KUKA KRL program: PrintBool.src

&ACCESS RVO
&PARAM EDITMASK = *
DEF PrintBool(name[]:in, value:in )
decl bool value
decl char name[]
decl KrlMsg_T msg
decl KrlMsgPar_T par[3]
decl KrlMsgOpt_T opt
decl int handle

msg = {modul[] "print", Nr 1, msg_txt[] "<bool> %1 = %2"}
par[1] = {par_type #value, par_txt[] " "}
par[1].par_txt[] = name[]
if value==true then
 par[2] = {par_type #value, par_txt[] "true"}
else
 par[2] = {par_type #value, par_txt[] "false"}
endif
opt = {vl_stop true, clear_p_reset true, clear_p_SAW false, log_to_DB false}
handle = Set_KrlMsg (#notify, msg, par[], opt)

END
